TYPE T_AnyInt : __SYSTEM.AnyType; END_TYPE

(* stored: Version 1.1.0.1
   DUT T_AnyInt: Id {75dd78c8-d5ac-45b1-a4bb-20c7a9c740ac} *)
